// TIA Portal V16 export
// export: Created 2022-11-14T17:35:40.7229198Z, ExportSetting WithDefaults, DisplayName Totally Integrated Automation Portal, DisplayVersion V16, DisplayName TIA Portal Version Control Interface, DisplayVersion V16, DisplayName TIA Portal Openness, DisplayVersion V16, DisplayName STEP 7 Professional, DisplayVersion V16, DisplayName STEP 7 Safety, DisplayVersion V16, DisplayName WinCC Advanced, DisplayVersion V16
DATA_BLOCK "DB08_Prestretch"   // DB8
{ S7_Optimized_Access := 'FALSE' }
AUTHOR : Robopac
VERSION : 0.0
// stored: AutoNumber false, IsOnlyStoredInLoadMemory false, IsWriteProtectedInAS false
   VAR RETAIN
      dbx0_0 : Bool := FALSE;   // Support memory for prestretch PGSM or PGSA
      dbx0_1 : Bool := FALSE;
      dbx0_2 : Bool := FALSE;
      dbx0_3 : Bool := FALSE;
      dbx0_4 : Bool := FALSE;
      dbx0_5 : Bool := FALSE;
      dbx0_6 : Bool := FALSE;
      dbx0_7 : Bool := FALSE;
      dbw2 : Int := 0;
      dbw4 : Int := 0;
      dbw6 : Int := 0;
      dbw8 : Int := 0;
      dbw10 : Int := 0;   // Film provided for every revolution at max speed (mm per revolution)
      dbw12 : Int := 0;   // Film force value to apply to pallet (mm)
      dbd14 : DInt := 0;   // Support memory for film force to apply to pallet
      dbw18 : Int := 0;   // Film force value to apply to pallet (analog value)
      dbw20 : Int := 0;   // Film force value to apply to pallet (%)
      dbw22 : Int := 0;
      dbw24 : Int := 0;
      dbw26 : Int := 0;
      dbw28 : Int := 0;
      dbw30 : Int := 0;   // Gain for analog scaling
      dbw32 : Int := 200;   // Film prestretch value to apply to pallet
      dbd34 : DInt := 0;   // Support memory for film prestretch to apply to pallet
      dbw38 : Int := 102;   // Film prestretch value to apply to pallet (analog value)
      dbw40 : Int := 0;
      dbw42 : Int := 0;
      dbw44 : Int := 0;
      dbw46 : Int := 0;
      dbw48 : Int := 0;
      dbw50 : Int := 0;   // Support for film prestretch test
      dbw52 : Int := 0;   // Support for film prestretch test
      dbw54 : Int := 0;   // Film weight every mm of film (10^-5 g/mm)
      dbw56 : Int := 0;
      dbw58 : Int := 0;
      dbw60 : Int := 0;
   END_VAR
BEGIN
END_DATA_BLOCK
